FUNCTION FC_CheckMinMaxReal : REAL		// Checks if the given value is within the min/max and if not will set either the MIN/MAX value
VAR_INPUT
	iValue:		REAL;
	iMin:		REAL;
	iMax:		REAL;
END_VAR

IF (iValue > iMax) THEN
	FC_CheckMinMaxReal := iMax;
ELSIF (iValue < iMin) THEN
	FC_CheckMinMaxReal := iMin;
ELSE
	FC_CheckMinMaxReal := iValue;
END_IF

END_FUNCTION

(* stored: Version 1.1.0.1, ProductVersion 3.1.4026.18
   POU FC_CheckMinMaxReal: Id {cc5606cf-b46f-4e7b-800a-557f48f2dbea}, SpecialFunc None *)
